TYPE csp_case_glue_ls_accU_lowerPosition_enum :
(
	CSP_CASE_GLUE_LS_ACCU_LOWERPOSITION_STATUS_NOT_INITIALIZED 									:= 0,
	CSP_CASE_GLUE_LS_ACCU_LOWERPOSITION_STATUS_DISABLED 										:= 10,
	CSP_CASE_GLUE_LS_ACCU_LOWERPOSITION_STATUS_POSITION_CHECK									:= 20,
	CSP_CASE_GLUE_LS_ACCU_LOWERPOSITION_STATUS_ENABLE_REQUEST 									:= 30,
	CSP_CASE_GLUE_LS_ACCU_LOWERPOSITION_STATUS_ENABLED 											:= 40,
	CSP_CASE_GLUE_LS_ACCU_LOWERPOSITION_STATUS_ABS_MOVE_REQUEST									:= 50,
	CSP_CASE_GLUE_LS_ACCU_LOWERPOSITION_STATUS_ABS_MOVING										:= 60,
	CSP_CASE_GLUE_LS_ACCU_LOWERPOSITION_STATUS_STOP_REQUEST 									:= 70,
	CSP_CASE_GLUE_LS_ACCU_LOWERPOSITION_STATUS_DISABLE_REQUEST 									:= 80,
	CSP_CASE_GLUE_LS_ACCU_LOWERPOSITION_STATUS_DISABLING 										:= 90
) := CSP_CASE_GLUE_LS_ACCU_LOWERPOSITION_STATUS_NOT_INITIALIZED;
END_TYPE

(* stored: Version 1.1.0.1, ProductVersion 3.1.4022.18
   DUT csp_case_glue_ls_accU_lowerPosition_enum: Id {daa72ac7-2772-4d3b-8a9b-bcb3964e1e77} *)
